RoboDK station: FUCKOFF.rdk

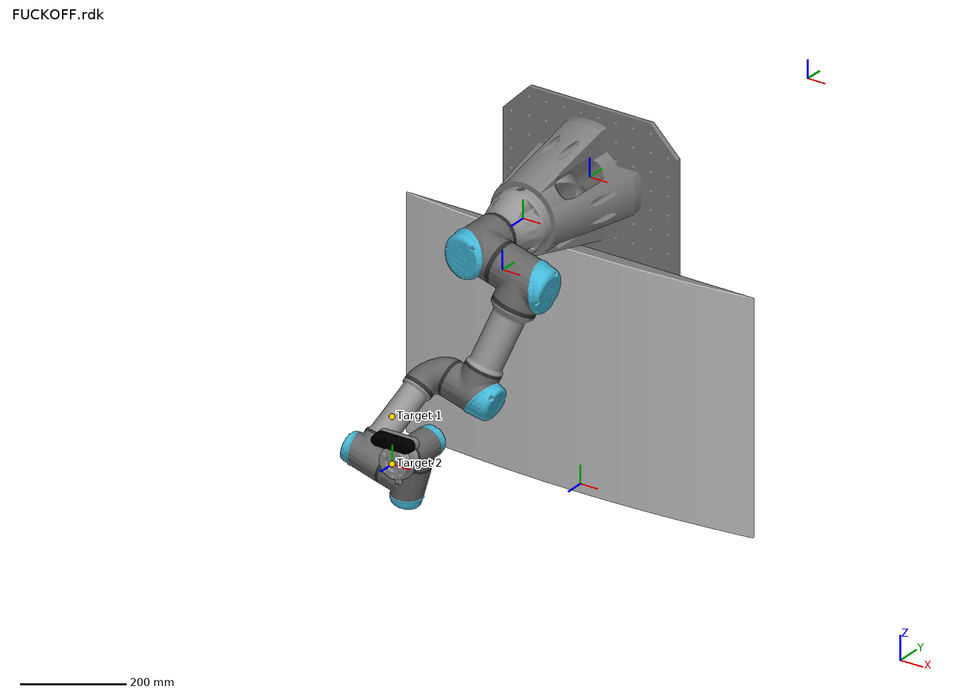
[picture v0: the station drawn from its stored meshes, robots at their saved joint values, targets as dots, program paths as lines]
Station FUCKOFF (saved by RoboDK 5.9.0). Poses are relative to the parent item; angles as X-Y-Z fixed-axis rotations.
Station parameters (name, value as stored): CollisionFreePlanner, UR3e, CollisionFreePlanner-Rob UR3e, LIN64
  - frame Frame 1 at (0, 0, 0) mm
    - object Bundplade at (0, 0, 0) mm, size 400 x 10 x 800 mm, geometry from Bundplade.stl
    - frame Frame 2 at (200, 0, 250) mm
      - object UR3e mount at (0, 0, 0) mm, size 239.9 x 218 x 239.9 mm, geometry from UR3e mount.stl
      - frame Frame 3 at (0, -218, 0) mm, rotated rx 90 ry 0 rz 0 deg
        - robot UR3e: 6 axes, payload 3 kg, reach 500 mm, repeatability 0.03 mm, weight 11 kg
            modified DH rows (alpha deg, a mm, theta deg, d mm): 0, 0, 0, 151.9; 90, 0, 180, 0; 0, 243.55, 0, 0; 0, 213.2, 0, 131.05; -90, 0, 0, 85.35; 90, 0, 180, 92.1
            joint limits [-360, -360, -360, -360, -360, -360] to [360, 360, 360, 360, 360, 360]; home [0, -90, -90, 0, 90, 0]; saved at [73.938, -21.6, -29.68, -218.72, 270, -163.938]
          - frame RealsenseHolder at (0, 0, 0) mm
            - object RealsenseHolder at (0, 0, -65) mm, size 90 x 104.9 x 9 mm, geometry from RealsenseHolder.stl
              - object RSD435 at (0, 44, 75) mm, size 90 x 25 x 25 mm, geometry from RSD435.stl
        - object Curve at (-50, -300, -150) mm
        - target Target 1 (Cartesian target) at (50, -200, 500) mm; joints [64.565, -10.134, -78.592, -181.274, 270, -154.565] of UR3e
        - target Target 2 (Cartesian target) at (50, -300, 500) mm; joints [73.938, -21.6, -29.68, -218.72, 270, -163.938] of UR3e
    - frame Frame 4 at (200, -30, -380) mm, rotated rx 90 ry 0 rz 0 deg
      - object TestpladeKurve v3 at (0, 0, -2973.5) mm, size 795.7 x 500 x 30.5 mm, geometry from TestpladeKurve v3.stl
  - frame UR3e Base at (0, 1000, 0) mm
  - camera Camera 1
  - program Target1ToTarget2 (3 instructions, listed below)
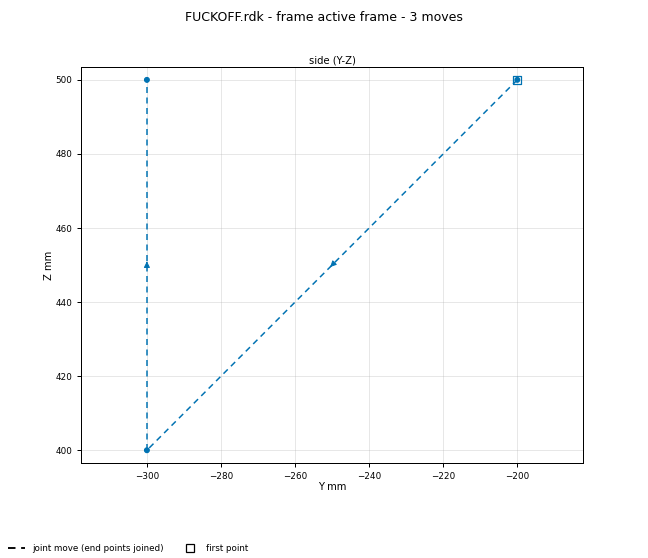
[picture p0: tool path of FUCKOFF.rdk in frame active frame, 3 of 3 moves have a stored position in this frame; points joined in program order, loops and branches not executed]

--- program Target1ToTarget2 (robot UR3e) ---
  MoveJ (Pt 1 (S9)) to (50, -200, 500) mm; joints [64.565, -10.134, -78.592, -181.274, 270, -154.565]
  MoveJ (Pt 2 (S15)) to (50, -300, 400) mm; joints [73.938, 5.197, -61.831, -213.366, 270, -163.938]
  MoveJ (Pt 3 (S18)) to (50, -300, 500) mm; joints [73.938, -21.6, -29.68, -218.72, 270, -163.938]
